TYPE NETWORK_BUFFER_SHORT :
STRUCT
	SIZE : UINT;
	BUFFER : NW_BUF_SHORT;
END_STRUCT
END_TYPE

(* stored: Version 1.1.0.1, ProductVersion 3.1.4024.4
   DUT NETWORK_BUFFER_SHORT: Id {acdcdf63-5d1b-4cb3-b194-af705ffa7e6c} *)
